# EPICS substitutions: vaccelApp/Db/power_converter.substitutions
file db/power_converter.rec
{
	pattern{ PC,     DEFAULT_CURRENT                     }
	#                2.44045585 / 1.1270572620311009e-02
               { Q1PDR,   216.5334390909285}
	#         	  2.44045585 / 1.1270572620311009e-02
               { Q1PTR,   216.5334390909285}

}
